PROGRAM Axis_02_Function_Blocks
VAR
END_VAR

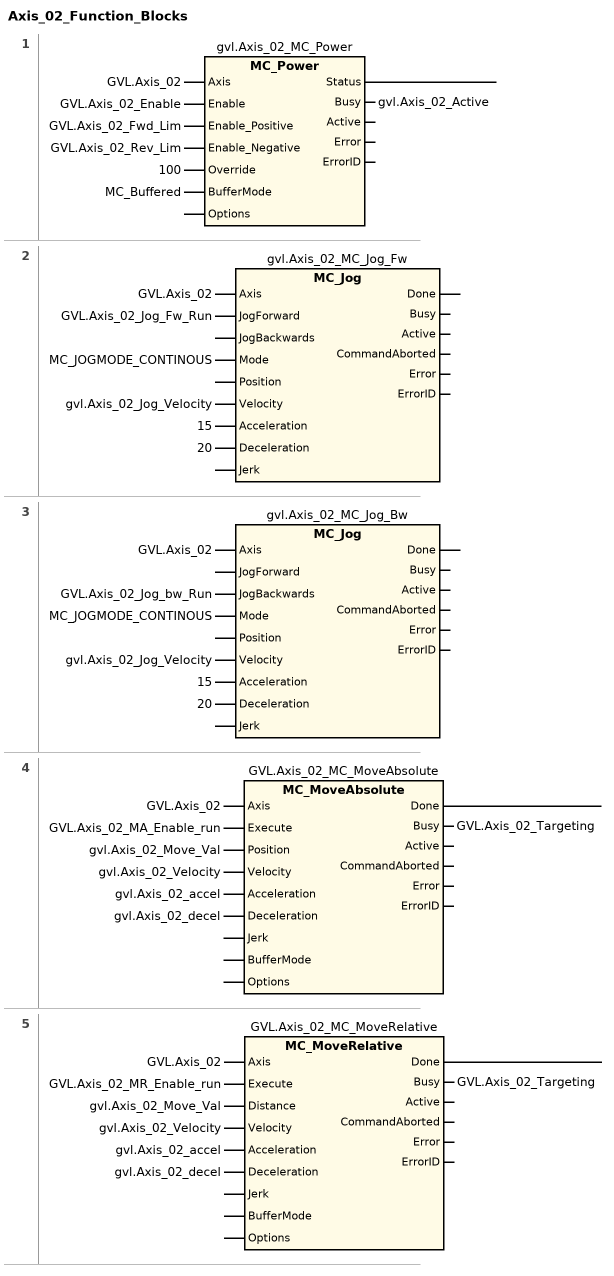
// NETWORK 1
gvl.Axis_02_MC_Power(
    Axis := GVL.Axis_02,
    Enable := GVL.Axis_02_Enable,
    Enable_Positive := GVL.Axis_02_Fwd_Lim,
    Enable_Negative := GVL.Axis_02_Rev_Lim,
    Override := 100,
    BufferMode := MC_Buffered,
    Busy => gvl.Axis_02_Active); // MC_Power

// NETWORK 2
gvl.Axis_02_MC_Jog_Fw(
    Axis := GVL.Axis_02,
    JogForward := GVL.Axis_02_Jog_Fw_Run,
    Mode := MC_JOGMODE_CONTINOUS,
    Velocity := gvl.Axis_02_Jog_Velocity,
    Acceleration := 15,
    Deceleration := 20); // MC_Jog

// NETWORK 3
gvl.Axis_02_MC_Jog_Bw(
    Axis := GVL.Axis_02,
    JogBackwards := GVL.Axis_02_Jog_bw_Run,
    Mode := MC_JOGMODE_CONTINOUS,
    Velocity := gvl.Axis_02_Jog_Velocity,
    Acceleration := 15,
    Deceleration := 20); // MC_Jog

// NETWORK 4
GVL.Axis_02_MC_MoveAbsolute(
    Axis := GVL.Axis_02,
    Execute := GVL.Axis_02_MA_Enable_run,
    Position := gvl.Axis_02_Move_Val,
    Velocity := gvl.Axis_02_Velocity,
    Acceleration := gvl.Axis_02_accel,
    Deceleration := gvl.Axis_02_decel,
    Busy => GVL.Axis_02_Targeting); // MC_MoveAbsolute

// NETWORK 5
GVL.Axis_02_MC_MoveRelative(
    Axis := GVL.Axis_02,
    Execute := GVL.Axis_02_MR_Enable_run,
    Distance := gvl.Axis_02_Move_Val,
    Velocity := gvl.Axis_02_Velocity,
    Acceleration := gvl.Axis_02_accel,
    Deceleration := gvl.Axis_02_decel,
    Busy => GVL.Axis_02_Targeting); // MC_MoveRelative

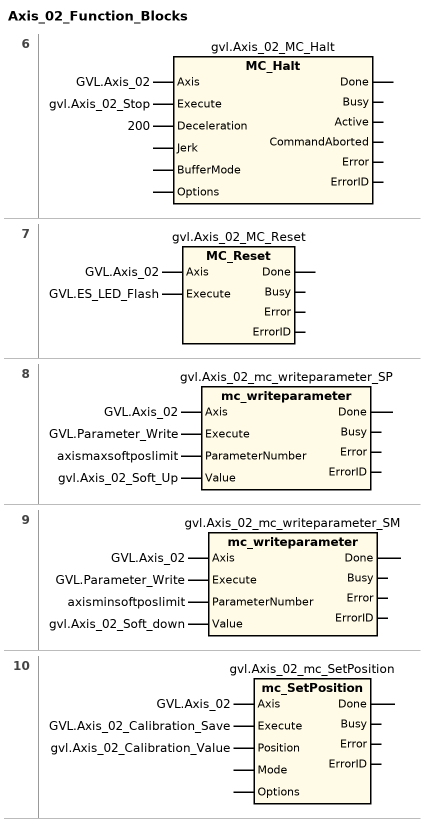
// NETWORK 6
gvl.Axis_02_MC_Halt(Axis := GVL.Axis_02, Execute := gvl.Axis_02_Stop, Deceleration := 200); // MC_Halt

// NETWORK 7
gvl.Axis_02_MC_Reset(Axis := GVL.Axis_02, Execute := GVL.ES_LED_Flash); // MC_Reset

// NETWORK 8
gvl.Axis_02_mc_writeparameter_SP(
    Axis := GVL.Axis_02,
    Execute := GVL.Parameter_Write,
    ParameterNumber := axismaxsoftposlimit,
    Value := gvl.Axis_02_Soft_Up); // mc_writeparameter

// NETWORK 9
gvl.Axis_02_mc_writeparameter_SM(
    Axis := GVL.Axis_02,
    Execute := GVL.Parameter_Write,
    ParameterNumber := axisminsoftposlimit,
    Value := gvl.Axis_02_Soft_down); // mc_writeparameter

// NETWORK 10
gvl.Axis_02_mc_SetPosition(
    Axis := GVL.Axis_02,
    Execute := GVL.Axis_02_Calibration_Save,
    Position := gvl.Axis_02_Calibration_Value); // mc_SetPosition

END_PROGRAM

(* stored: Version 1.1.0.1, ProductVersion 3.1.4022.12
   POU Axis_02_Function_Blocks: Id {aa037c8e-11fc-476e-a077-f1731c2fb5ae}, SpecialFunc None *)
